# EPICS autosave request: usbApp/Db/LogitechF710_settings.req
file UserSeq.req P=$(P),R=$(R),SEQ=UpSeq
file UserSeq.req P=$(P),R=$(R),SEQ=DownSeq
file UserSeq.req P=$(P),R=$(R),SEQ=LeftSeq
file UserSeq.req P=$(P),R=$(R),SEQ=RightSeq

file UserSeq.req P=$(P),R=$(R),SEQ=LSUpSeq
file UserSeq.req P=$(P),R=$(R),SEQ=LSDownSeq
file UserSeq.req P=$(P),R=$(R),SEQ=LSLeftSeq
file UserSeq.req P=$(P),R=$(R),SEQ=LSRightSeq

file UserSeq.req P=$(P),R=$(R),SEQ=RSUpSeq
file UserSeq.req P=$(P),R=$(R),SEQ=RSDownSeq
file UserSeq.req P=$(P),R=$(R),SEQ=RSLeftSeq
file UserSeq.req P=$(P),R=$(R),SEQ=RSRightSeq

file UserSeq.req P=$(P),R=$(R),SEQ=ASeq
file UserSeq.req P=$(P),R=$(R),SEQ=BSeq
file UserSeq.req P=$(P),R=$(R),SEQ=XSeq
file UserSeq.req P=$(P),R=$(R),SEQ=YSeq

file UserSeq.req P=$(P),R=$(R),SEQ=LTSeq
file UserSeq.req P=$(P),R=$(R),SEQ=LBSeq
file UserSeq.req P=$(P),R=$(R),SEQ=RTSeq
file UserSeq.req P=$(P),R=$(R),SEQ=RBSeq
file UserSeq.req P=$(P),R=$(R),SEQ=L3Seq
file UserSeq.req P=$(P),R=$(R),SEQ=R3Seq
